FUNCTION_BLOCK FB_SIM_MICADO_PUMPS
VAR_INPUT
	in_RefPVP:	REFERENCE TO FB_CRYO_PUMP_ECODRY;
	in_RefTMP:	REFERENCE TO FB_CRYO_PUMP_ATH2303M;
	in_Delay:	TIME := T#10S;
END_VAR
VAR_OUTPUT
END_VAR
VAR
	trgStart_PVP:	R_TRIG;
	trgStart_TMP:	R_TRIG;
	trgStop_PVP:	F_TRIG;
	trgStop_TMP:	F_TRIG;
	
	timer_PVP:		TON;
	timer_TMP:		TON;
	
	bON_PVP:		BOOL := FALSE;
	bON_TMP:		BOOL := FALSE;
	
	q_PVP_Running	AT %Q*:	BOOL := TRUE;	// Active low!
	q_TMP_Ready		AT %Q*:	BOOL;
	q_TMP_Speed100	AT %Q*:	BOOL;
	
	ptrTMP_Speed:	POINTER TO DINT;
END_VAR

// Assign pointer to TMP speed.
ptrTMP_Speed	:= ADR(in_RefTMP.stat.nPumpSpeed);

// Get Start signals
trgStart_PVP(CLK:=in_RefPVP.in_bEnable);
trgStart_TMP(CLK:=in_RefTMP.in_bEnable);

// Get Stop signals
trgStop_PVP(CLK:=in_RefPVP.in_bEnable);
trgStop_TMP(CLK:=in_RefTMP.in_bEnable);

// Start timer on Start/Stop events
IF trgStart_PVP.Q THEN
	bON_PVP	:= TRUE;
	timer_PVP(IN:=FALSE);
	timer_PVP(IN:=TRUE, PT:=in_Delay/2);
ELSIF trgStop_PVP.Q THEN
	bON_PVP	:= FALSE;
	timer_PVP(IN:=FALSE);
	timer_PVP(IN:=TRUE, PT:=in_Delay/2);
END_IF

IF trgStart_TMP.Q THEN
	bON_TMP	:= TRUE;
	timer_TMP(IN:=FALSE);
	timer_TMP(IN:=TRUE, PT:=in_Delay);
ELSIF trgStop_TMP.Q THEN
	bON_TMP	:= FALSE;
	timer_TMP(IN:=FALSE);
	timer_TMP(IN:=TRUE, PT:=in_Delay * 2);
END_IF

// Execute timers
timer_PVP();
timer_TMP();

// Set outputs on timer expiry
IF timer_PVP.Q THEN
	// NOTE: PVP feedback is active low.
	IF bON_PVP THEN
		q_PVP_Running	:= FALSE;
	ELSE
		q_PVP_Running	:= TRUE;
	END_IF
END_IF

IF bON_TMP  AND (NOT timer_TMP.Q AND timer_TMP.ET > T#3S) THEN
	// Starting up.
	// Set speed > 100 rpm after 3 sec.
	ptrTMP_Speed^	:= 500;
	q_TMP_Speed100	:= TRUE;
END_IF

IF NOT bON_TMP  AND (NOT timer_TMP.Q AND timer_TMP.ET > T#5S) THEN
	// Stopping the pump.
	// Not ready after 5 sec.
	// However, the pump is still spinning.
	ptrTMP_Speed^	:= 1800;
	q_TMP_Ready		:= FALSE;
END_IF

IF timer_TMP.Q THEN
	IF bON_TMP THEN
		ptrTMP_Speed^	:= 2000;
		q_TMP_Ready	:= TRUE;
	ELSE
		ptrTMP_Speed^	:= 0;
		q_TMP_Ready		:= FALSE;
		q_TMP_Speed100	:= FALSE;
	END_IF
END_IF

END_FUNCTION_BLOCK

(* stored: Version 1.1.0.1, ProductVersion 3.1.4024.10
   POU FB_SIM_MICADO_PUMPS: Id {e34ea3d5-f755-420e-95b8-32ab710aaa31}, SpecialFunc None *)
